(* CoDeSys 2.3 export: FB_PERSISTENT.EXP *)

(* POU FB_Persistent, FBD *)
FUNCTION_BLOCK FB_Persistent

(*********************************************************************************************************************************)
(*								Beckhoff Automation Poland												*)
(* 									FB_Persistent 	v1.5												*)
(* 										20.08.2014														*)
(* 							v1.5 - zmiana minimalnego interwalu zapisu									*)
(* 					Blok funkcyjny zapisujący zmienne typu persistent na karcie CF						*)
(* 						Możliwy zapis na żądanie lub z określoną częstotliwością.  						*)
(* 				Pozostawienie wejscia tInterval bez zmiennej wyłacza funkcję zapisu cyklicznego			*)
(* 							Minimalny czas między zapisem cyklicznym 30s								*)
(* 				Konieczne jest dodanie biblioteki TcUtilities.lib, TcSystem.lib oraz TcBase.lib					*)
(*			 UWAGA: Blok przygotowany dla RunTime 1 port 801 - typowa konfiguracja 					*)
(*_____________________________________________________________________________________*)

VAR_INPUT
	bWrite			: BOOL;							(*Zapis na rozkaz *)
	tInterval			: TIME:=T#71582m47s295ms;		(*Czestotliwosc zapisu na karte CF*)
END_VAR
VAR_OUTPUT
	bBusy			: BOOL;
	bErr			: BOOL;
	udErrID			: UDINT;
END_VAR
VAR
	fbWritePersistentData	: FB_WritePersistentData; 	(* Blok zapisu *)
	t1						: TON;						(* Timer zapisu *)
	_GETCURTASKINDEX	: GETCURTASKINDEX;		(* Informacja o Tasku *)
	BIndex					: BYTE;						(* Nr tasku *)
END_VAR
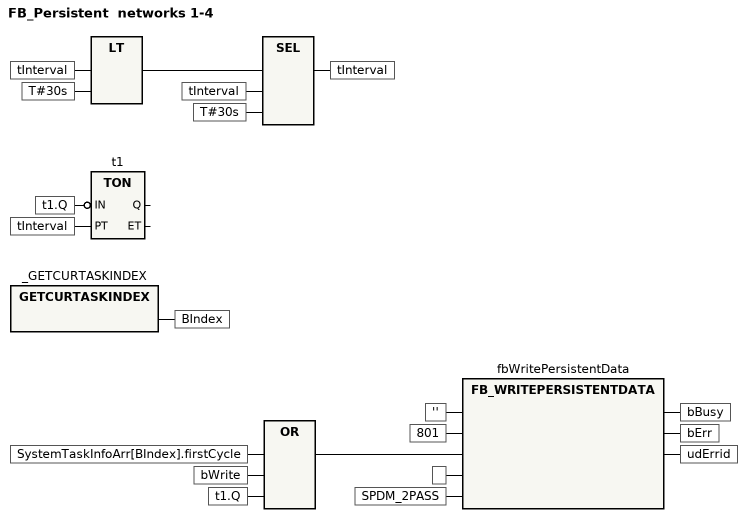
_FBD_ (* Function Block Diagram *)
NETWORK 1 (* Comment: Zabezpieczenie karty - czestotliwosc zapisu nie moze byc mniejsza niz 30s *)
	SEL(LT(tInterval, T#30s), tInterval, T#30s) => tInterval
NETWORK 2 (* Comment: Wyzwalanie zapisu *)
	t1:TON(IN: NOT t1.Q, PT: tInterval)
NETWORK 3
	_GETCURTASKINDEX:GETCURTASKINDEX() => BIndex
NETWORK 4 (* Comment: Blok zapisu *)
	fbWritePersistentData:FB_WRITEPERSISTENTDATA('', 801, OR(SystemTaskInfoArr[BIndex].firstCycle, bWrite, t1.Q), , SPDM_2PASS, out 2 => bErr, out 3 => udErrid) => bBusy
_END_FBD_
(* the same logic as Structured Text *)
(* Network 1 *)
tInterval := SEL(tInterval < T#30s, tInterval, T#30s);
(* Network 2 *)
t1(IN := NOT t1.Q, PT := tInterval);
(* Network 3: see the listing above *)
(* Network 4: see the listing above *)
END_FUNCTION_BLOCK
